FUNCTION_BLOCK FB_Test_Component EXTENDS FB_FCSLComponentBase IMPLEMENTS I_TestComponent

VAR
	_trig : BOOL;
	Trig : R_TRIG;
	_trig2 : BOOL;
	Trig2 : R_TRIG;
END_VAR

VAR
	// Inputs
	MyInput AT %I* : BOOL;

	// Outputs
	MyOutput AT %Q* : BOOL;

	// HMI
//	MyComponent_HMI			: ST_ComponentMyComponent_HMI;
//	HMICommandDescendant_RT : R_TRIG;

	// Alarms
//	MyComponentAlarms : ARRAY[1..MY_COMPONENT_ALARMS_COUNT] OF FB_TcAlarm;

	// Internal variables
//	_MyVarProperty1 : BOOL;
//	_MyVarProperty2 : BOOL;
//	MyVarInternal1	: BOOL;
//	MyVarInternal2	: BOOL;

	//MyCommandFb		: MyCommandFB;// Command FB to execute something e.g. MC_MoveAbsolute
END_VAR

VAR CONSTANT
//	MY_COMPONENT_ALARMS_COUNT : UDINT := 2;
END_VAR

// NO CODE HERE!!!

//! @summary Basic component initialization logic
METHOD CyclicLogic

//! @description This method is called by <c>CyclicLogic()</c> as required
//! @description This method should be called cyclically by descendant function blocks by invoking <c>SUPER^.CyclicLogic()</c>. 
// Alternatively, the contents of this method could be reimplemented entirely in which case a call to this method would not be necessary.

VAR
END_VAR
IF NOT _InitComplete THEN
	_InitComplete := Initialize();
	RETURN;
END_IF

//{error 'Programming instruction - Write your custom component cyclic cogic here'}

Trig(CLK := _trig);
Trig2(CLK := _trig2);

IF Trig.Q THEN
	M_SysLog(msg := CONCAT(Name, ' : Has being triggered 1'), debug := E_SysLogLevel.testing);
END_IF

IF Trig.Q THEN
	M_SysLog(msg := CONCAT(Name, ' : Has being triggered 2'), debug := E_SysLogLevel.testing);
END_IF
IF Trig2.Q THEN
	M_AuditLog(k := 'Login', v := 'User 1234 has logged in');
END_IF

(*
	MyCommandFb();
	IF MyCommandFB.Error THEN
		_Error	 := TRUE;
		_ErrorID := MyCommandFb.ErrorId;
	END_IF
	
	MyCommandFB.Execute := FALSE;
*)

// Component Error
//{error 'Programming instruction - Create component has error'}
//_Error	 := TRUE;
//_ErrorID := 9999;

// Component Busy
//{error 'Programming instruction - Create component is busy'}
IF FALSE THEN
	_Busy := TRUE;
ELSE
	_Busy := FALSE;
END_IF

// Call Super
SUPER^.CyclicLogic();

// Set Current Alarm Severity
// _CurrentAlarmSeverity := F_GetMaxSeverityRaised(Alarms := MyComponentAlarms, CurrentSeverity := _CurrentAlarmSeverity);
END_METHOD

(*! @summary Basic component initialization logic*)
METHOD PROTECTED Initialize : BOOL
// TODO : {error 'Programming instruction - Add code to initialize your Component'}
//M_SysLog(msg := CONCAT(Name, ' : Has being initalized'), debug := E_SysLogLevel.production);

// Call Super
Initialize := Super^.Initialize();
END_METHOD

PROPERTY pTrig : BOOL
GET
pTrig := _trig;
END_GET
SET
_trig := pTrig;
END_SET
END_PROPERTY

PROPERTY pTrig2 : BOOL
GET
pTrig2 := _trig2;
END_GET
SET
_trig2 := pTrig2;
END_SET
END_PROPERTY

END_FUNCTION_BLOCK

(* stored: Version 1.1.0.1
   POU FB_Test_Component: Id {80924ee2-d833-4cc9-a197-975646d7a2bc}, SpecialFunc None
   Folder I_CyclicLogic: Id {949d3941-c769-4ef9-9270-365ad2e53f9d}
   Folder Methods: Id {785d2a36-efb8-4cbd-9276-380be6e85a49}
   Method CyclicLogic: Id {1d14c55b-7a16-4bb6-af0b-ba890cf004a4}
   Method Initialize: Id {f036e164-e0c3-48f7-be80-28e215b37540}
   Property pTrig: Id {6000d349-0d03-40cb-ae39-d4afc417b620}
   Get Get: Id {9029c822-5889-40b9-a98b-b42ee0c4ef21}
   Set Set: Id {31a903c1-e28c-4057-a4d5-690594455fca}
   Property pTrig2: Id {bff14ddd-be64-430c-bab9-53d8c94a9042}
   Get Get: Id {a300b180-cc1e-4b95-a88c-8654a9b58184}
   Set Set: Id {1df91c02-74bd-4908-8347-9e3dbfa6784e} *)
